// TwinCAT 3 PLC project PLCProgram
// ProgramVersion: 3.1.4026.24
// libraries:
//   FactoryIO_Library, * (Privat)
//   Tc2_ModbusSrv, * (Beckhoff Automation GmbH)
//   Tc2_Standard, * (Beckhoff Automation GmbH)
//   Tc2_System, * (Beckhoff Automation GmbH)
//   Tc2_Utilities, * (Beckhoff Automation GmbH)
// project tree:
//   DUTs/Program/OrderManagement/ OrderData.TcDUT, OrderType.TcDUT
//   DUTs/Program/RFID/ DataPositions.TcDUT
//   DUTs/Program/Warehouse/ StackerCraneStepsLoading.TcDUT, StackerCraneStepsUnloading.TcDUT
//   GVLs/ ConveyorbeltsInfeed.TcGVL, ConveyorbeltsOutfeed.TcGVL, Emitter.TcGVL, GVL.TcGVL, OperatingMode.TcGVL, HMI.TcGVL, OrderManagement.TcGVL, Remover.TcGVL, RFID.TcGVL, Signalmapping.TcGVL, Warehouse.TcGVL
//   / PlcTask.TcTTO
//   POUs/ MAIN.TcPOU, SignalmappingInput.TcPOU, SignalmappingOutput.TcPOU
//   POUs/Programm/AdditionalFunctions/RunControl/ FB_RunControl.TcPOU
//   POUs/Programm/General/ Call_HMI.TcPOU, Call_Operatingmode.TcPOU
//   POUs/Programm/Sections/Infeed/ Call_ConveyorbeltsInfeed.TcPOU, Call_Emitter.TcPOU, Call_RFID.TcPOU
//   POUs/Programm/Sections/Outfeed/ Call_ConveyorbeltsOutfeed.TcPOU, Call_Remover.TcPOU
//   POUs/Programm/Sections/Warehouse/ Call_OrderManagement.TcPOU, Call_Warehouse.TcPOU
// real-time tasks:
//   TASK PlcTask: cycle T#10ms, priority 20, ADS port 350

CONFIGURATION PLCProgram
    RESOURCE PLC ON TwinCAT3
        TASK PlcTask(INTERVAL := T#10ms, PRIORITY := 20);
        PROGRAM MAIN WITH PlcTask : MAIN;
    END_RESOURCE
END_CONFIGURATION

// ---- DUTs/Program/OrderManagement/OrderData.TcDUT
TYPE OrderData :
STRUCT
	JobType	:	OrderType;	//Kind of Order; None, Loading, Unloading
	WarehousePlace	:	WORD;	//Place in the warehouse whre part should be picked or put
	SerialNumberItem	:	WORD;	//Serialnumber of the part
	OrderDone	:	BOOL;	//Current order is finished
	NewOrderSend	:	BOOL;	//Order application has sent new order
	NewOrderReceived	:	BOOL;	//PLC has received new data
END_STRUCT
END_TYPE

// ---- DUTs/Program/OrderManagement/OrderType.TcDUT
{attribute 'qualified_only'}
{attribute 'strict'}
{attribute 'to_string'}
TYPE OrderType :
(
	None := 0,
	Loading,
	Unloading
);
END_TYPE

// ---- DUTs/Program/RFID/DataPositions.TcDUT
TYPE DataPositions :
STRUCT
	FeedInReadingPoint	:	WORD;
	FeedInStackerCrane	:	WORD;
	StackerCraneFork	:	WORD;
END_STRUCT
END_TYPE

// ---- DUTs/Program/Warehouse/StackerCraneStepsLoading.TcDUT
{attribute 'qualified_only'}
{attribute 'strict'}
{attribute 'to_string'}
TYPE StackerCraneStepsLoading :
(
	Waiting := 0,
	DriveToLoadingPosition,
	ForkUnderLoad,
	LiftLoadItem,
	ForkToMiddle,
	DriveToUnloadPrePosition,
	ForkInWarehouse,
	DriveToUnloadPosition
);
END_TYPE

// ---- DUTs/Program/Warehouse/StackerCraneStepsUnloading.TcDUT
{attribute 'qualified_only'}
{attribute 'strict'}
{attribute 'to_string'}
TYPE StackerCraneStepsUnloading :
(
	Waiting := 0,
	DriveToWarehousePlace,
	ForkInWarehouse,
	LiftPart,
	ForkToMiddle,
	DriveToUnloadingPlace,
	ForkToRight,
	LowerPart
);
END_TYPE

// ---- GVLs/ConveyorbeltsInfeed.TcGVL
VAR_GLOBAL
	instConveyorFeedIn	:	FactoryIO.FB_Foerderband;
	instConveyorFeedInStackerCrane	:	FactoryIO.FB_Foerderband;
	conFdIRunControlForwardActiv	:	BOOL;	//Runcontrol forward activ
	conFdIStCRunControlForwardActiv	:	BOOL;	//Runcontrol forward activ
	feConveyorInfeedEnd	:	F_TRIG;	//Falling edge sensor end conveyor infeed
END_VAR

// ---- GVLs/ConveyorbeltsOutfeed.TcGVL
VAR_GLOBAL
	instConveyorFeedOutStackerCrane	:	FactoryIO.FB_Foerderband;
	instConveyorFeedOutTwoMeter	:	FactoryIO.FB_Foerderband;
	instConveyorFeedOutCurve	:	FactoryIO.FB_Foerderband;
	instConveyorFeedOutLong	:	FactoryIO.FB_Foerderband;
	instPartMovingOut	:	FB_RunControl;
END_VAR

// ---- GVLs/Emitter.TcGVL
VAR_GLOBAL
	instEmitterConveyorFeedIn	:	FactoryIO.FB_Emitter;	//Instanz FB_Emitter Zufuehrband Einlauf
	
END_VAR

// ---- GVLs/GVL.TcGVL
{attribute 'qualified_only'}
VAR_GLOBAL
	//Hier die Array-Grenzen anpassen auf die maximale Anzahl an Signalen.
	//Der Name der Liste, darf nicht verändert werden.
	mb_Input_Coils        : ARRAY [0..255] OF BOOL;	//Digital outputs of the PLC
    mb_Output_Coils       : ARRAY [0..255] OF BOOL;	//Digital inputs of the PLC
    mb_Input_Registers    : ARRAY [0..255] OF WORD;	//Analog outputs of the PLC
    mb_Output_Registers   : ARRAY [0..255] OF WORD;	//Analog inputs of the PLC	
END_VAR

// ---- GVLs/OperatingMode.TcGVL
VAR_GLOBAL
	instOperatingmode	:	FactoryIO.FB_OperatingMode;
	currentStateOperatingMode	:	FactoryIO.OperatingMode;
	permissionHardware	:	BOOL := TRUE;
	permissionSafety	:	BOOL := TRUE;
END_VAR

// ---- GVLs/HMI.TcGVL
VAR_GLOBAL
	hmiHeaderInstance	:	FB_HMIHeader;
	hmiHeaderInterface	:	HMIHeader;	
	hmiOperatingmodeInterface	:	HMIInterfaceOperatingMode;
	
	hmiAdsCommunicationInterfaceInstance	:	FB_ADSCommunicationStatus;
	hmiAdsCommunicationInterface	:	ADSCommunicationInterface;
	
	hmiMachineSectionInterface	:	MachineSectionHMIInterface;
	
	hmiEmitterInstances	:	ARRAY[0..0] OF STRING := [
														'FeedIn'
													];
	hmiConveyorInstances	:	ARRAY[0..5] OF STRING := [
															'FeedIn',
															'FeedIn StackerCrane',
															'FeedOut StackerCrane',
															'FeedOut Two meter',
															'FeedOut Curve',
															'FeedOut long'
														 ];
	hmiStackerCraneInstances	:	ARRAY[0..0] OF STRING := [
															'StackerCrane'
														 ];		
	hmiRFIDInstances	:	ARRAY[0..0] OF STRING := [
															'FeedIn StackerCrane'
														 ];
	hmiRemoverInstances	:	ARRAY[0..0] OF STRING := [
														'FeedOut'
													];
END_VAR

// ---- GVLs/OrderManagement.TcGVL
VAR_GLOBAL
	currentOrderData	:	OrderData;
	nextJobReady	:	BOOL;
	reOrderDone	:	R_TRIG;
	reNewOrderSend	:	R_TRIG;
	reShiftSerialNumber	:	R_TRIG;
END_VAR

// ---- GVLs/Remover.TcGVL
VAR_GLOBAL
	ConveyorFeedOutLongRemover	:	BOOL;	//Conveyor feed out long remover
	instRemoverConveyorOutfeedLong	: FactoryIO.FB_Remover;	//Instance of FB_Remover
END_VAR

// ---- GVLs/RFID.TcGVL
VAR_GLOBAL
	instRFIDInfeed	:	FactoryIO.FB_RFID;	//Instance of the RFID-Sensor
	finishedMessageReadSerialNumber	:	BOOL;
	reReadSerialNumber	:	R_TRIG;
	reFinishedMessageReadSerialNumber	:	R_TRIG;
	readData	:	DataPositions;
END_VAR

// ---- GVLs/Signalmapping.TcGVL
VAR_GLOBAL
	BA_Manuel	:	BOOL;	//Operatingmode manual
	BA_Automatik	:	BOOL;	//Operatingmode automatic
	NotAus_Hochregallager	:	BOOL;	//E_Stop
	Start_Automatik_Hochregallager	:	BOOL;	//Automatic Start
	Stop_Automatik_Hochregallager	:	BOOL;	//Automatic Stop
	Grundstellung_Automatik_Hochregallager	:	BOOL;	//Homing
	Reset_Hochregallager	:	BOOL;	//Reset
	Quit_Hochregallager	:	BOOL;	//Quit
	PartPresentConveyorInfeedBegin	:	BOOL;	//Sensor Emitter part present
	PartPresentConveyorInfeedEnd	:	BOOL;	//Sensor conveyor feed in part present
	PartPresentConveyorInfeedStCEnd	:	BOOL;	//Sensor conveyor feed in stacker crane part present
	StackerCraneOneXAxisIsMoving	:	BOOL;	//Stacker crane X axis is moving
	StackerCraneOneZAxisIsMoving	:	BOOL;	//Stacker crane Z axis is moving
	Gabel_InPos_Links	:	BOOL;	//Stacker crane fork in pos left
	Gabel_InPos_Mitte	:	BOOL;	//Stacker crane fork in pos middle
	Gabel_InPos_Rechts	:	BOOL;	//Stacker crane fork in pos right
	SensorConveyorOutfeedStackerCrane	:	BOOL;	//Sensor conveyor feed out stacker crane part present
	SensorConveyorOutfeedEnd	:	BOOL;	//Sensor conveyor feed out part present
	Button_Start_LED	:	BOOL;	//LED start button
	Button_Stop_LED	:	BOOL;	//LED stop button
	Button_Grundstellung_LED	:	BOOL;	//LED homing button
	Button_Reset_LED	:	BOOL;	//LED reset button
	Button_Quit_LED	:	BOOL;	//LED quit button
	EmitterFeedIn	:	BOOL;	//Emitter
	FeedInForward	:	BOOL;	//Conveyor feed in forward
	FeedInStackerCraneForward	:	BOOL;	//Conveyor feed in stacker crane forward
	RFIDFeedInExecuteCommand	:	BOOL;	//RFID feed in stacker crane execute command
	Gabel_zu_Pos_Links	:	BOOL;	//Stacker crane fork left
	Gabel_zu_Pos_Rechts	:	BOOL;	//Stacker crane fork right
	StackerCraneOneLiftFork	:	BOOL;	//Stacker crane lift fork
	ConveyorFeedOutStackerCrane	:	BOOL;	//Conveyor feed out stacker crane forward
	ConveyorFeedOutTwoMeter  	:	BOOL;	//Conveyor feed out forward
	ConveyorCurveFeedOut  	:	BOOL;	//Conveyor curvefeed out forward
	ConveyorFeedOutLong  	:	BOOL;	//Conveyor feed out long forward
	RFIDFeedInReceivedCommandID	:	WORD;	//RFID feed in stacker crane feedback command ID
	RFIDFeedInStatus	:	WORD;	//RFID feed in stacker crane status
	RFIDFeedInReadData	:	WORD;	//RFID feed in stacker crane read data
	RFIDFeedInCommand	:	WORD;	//RFID stacker crane feed in command
	RFIDFeedInMemoryIndex	:	WORD;	//RFID stacker crane feed in memory index
	RFIDFeedInWriteData	:	WORD;	//RFID stacker crane feed in data write
	StackerCraneOneTargetPos  	:	WORD;	//Stacker crane one index position
END_VAR

// ---- GVLs/Warehouse.TcGVL
VAR_GLOBAL
	InUnloading	:	BOOL;
	PartPresent	:	BOOL;
	LoadingSequenceActive	:	BOOL;
	UnloadingSequenceActive	:	BOOL;
	instStackerCrane	:	FB_StackerCrane_Numerical;
	processStepsLoading	: StackerCraneStepsLoading;	
	processStepsUnloading	: StackerCraneStepsUnloading;
	LiftLowerPartLoadingprocess	:	TON;
	LiftLowerPartUnloadingprocess	:	TON;
END_VAR

// ---- POUs/MAIN.TcPOU
PROGRAM MAIN
VAR
	
END_VAR

SignalmappingInput();
Call_Operatingmode();
Call_HMI();
Call_Emitter();
Call_ConveyorbeltsInfeed();
Call_RFID();
Call_OrderManagement();
Call_Warehouse();
Call_ConveyorbeltsOutfeed();
Call_Remover();
SignalmappingOutput();

END_PROGRAM

// ---- POUs/SignalmappingInput.TcPOU
FUNCTION SignalmappingInput

(*=============== Digitale Eingaenge ===============*)
BA_Manuel	:=	GVL.mb_Output_Coils[0];
BA_Automatik	:=	GVL.mb_Output_Coils[1];
NotAus_Hochregallager	:=	GVL.mb_Output_Coils[2];
Start_Automatik_Hochregallager	:=	GVL.mb_Output_Coils[3];
Stop_Automatik_Hochregallager	:=	GVL.mb_Output_Coils[4];
Grundstellung_Automatik_Hochregallager	:=	GVL.mb_Output_Coils[5];
Reset_Hochregallager	:=	GVL.mb_Output_Coils[6];
Quit_Hochregallager	:=	GVL.mb_Output_Coils[7];
PartPresentConveyorInfeedBegin	:=	GVL.mb_Output_Coils[9];
PartPresentConveyorInfeedEnd	:=	GVL.mb_Output_Coils[10];
PartPresentConveyorInfeedStCEnd	:=	GVL.mb_Output_Coils[11];
StackerCraneOneXAxisIsMoving	:=	GVL.mb_Output_Coils[13];
StackerCraneOneZAxisIsMoving	:=	GVL.mb_Output_Coils[14];
Gabel_InPos_Links	:=	GVL.mb_Output_Coils[15];
Gabel_InPos_Rechts	:=	GVL.mb_Output_Coils[16];
Gabel_InPos_Mitte	:=	GVL.mb_Output_Coils[17];
SensorConveyorOutfeedStackerCrane	:=	GVL.mb_Output_Coils[19];
SensorConveyorOutfeedEnd	:=	GVL.mb_Output_Coils[20];

(*=============== Analoge Eingaenge ===============*)
RFIDFeedInReceivedCommandID	:=	GVL.mb_Output_Registers[3];
RFIDFeedInStatus	:=	GVL.mb_Output_Registers[4];
RFIDFeedInReadData	:=	GVL.mb_Output_Registers[5];

END_FUNCTION

// ---- POUs/Programm/General/Call_Operatingmode.TcPOU
FUNCTION Call_Operatingmode

instOperatingmode(PermissionHardware := permissionHardware,
				  PermissionSoftware := permissionSafety,
				  E_Stop := NotAus_Hochregallager,
				  OperatingModeManual:= BA_Manuel, 
				  OperatingModeAutomatic:= BA_Automatik, 
				  HMIInterface := hmiOperatingmodeInterface,
				  LEDStart=> Button_Start_LED, 
				  LEDStop=> Button_Stop_LED, 
				  LEDHome=> Button_Grundstellung_LED, 
				  LEDReset=> Button_Reset_LED, 
				  LEDQuit=> Button_Quit_LED);

instOperatingMode.Start_On(Start_Automatik_Hochregallager);
instOperatingMode.Stop_On(Stop_Automatik_Hochregallager);
instOperatingMode.Homeing_On(Grundstellung_Automatik_Hochregallager);
instOperatingMode.Reset_On(Reset_Hochregallager);
instOperatingMode.Quit_On(Quit_Hochregallager);

currentStateOperatingMode := instOperatingmode.StateOperatingMode;

END_FUNCTION

// ---- POUs/Programm/General/Call_HMI.TcPOU
FUNCTION Call_HMI

hmiHeaderInstance(NameApplication := 'Hochregallager',
				  OperatingModeHMIInterface := hmiOperatingmodeInterface,
				  HeaderHMIInterface := hmiHeaderInterface);
			  
hmiAdsCommunicationInterfaceInstance(Timeout := T#1S,
									 TimeoutHMI := T#500ms,
									 LocalAdsPort := 851,
									 HeartbeatHMI := hmiAdsCommunicationInterface.HeartbeatHMI);
									 

hmiAdsCommunicationInterface.DeviceIpAddress := hmiAdsCommunicationInterfaceInstance.LocalIpAddress;
hmiAdsCommunicationInterface.LocalAMSNetId := hmiAdsCommunicationInterfaceInstance.LocalAMSNetId;
hmiAdsCommunicationInterface.HeartbeatPLC := hmiAdsCommunicationInterfaceInstance.PLCHeartbeatHMICommunication;
hmiAdsCommunicationInterface.RuntimeStatus := hmiAdsCommunicationInterfaceInstance.AdsState;

END_FUNCTION

// ---- POUs/Programm/Sections/Infeed/Call_Emitter.TcPOU
FUNCTION Call_Emitter
VAR_INPUT
END_VAR
VAR
END_VAR

instEmitterConveyorFeedIn(PartPresent:= PartPresentConveyorInfeedBegin, 
					   	  ActorInstanceIndex := 0,
					   	  ActorInstanceName := 'FeedIn',
					   	  HMIInterface := hmiMachineSectionInterface,
					   	  CreatePart=> EmitterFeedIn);
					   
IF NOT PartPresentConveyorInfeedBegin AND 
	currentStateOperatingMode.AutomaticStart.IsActive
THEN
	instEmitterConveyorFeedIn.Create();
END_IF

END_FUNCTION

// ---- POUs/Programm/Sections/Infeed/Call_ConveyorbeltsInfeed.TcPOU
FUNCTION Call_ConveyorbeltsInfeed

(*================ FeedIn ================*)
instConveyorFeedIn(
	SensorInfeed:= PartPresentConveyorInfeedBegin, 
	SensorOutfeed:= PartPresentConveyorInfeedEnd, 
	MaximumTimeRuncontrol:= T#30S, 
	ActorInstanceIndex := 0,
	ActorInstanceName := 'FeedIn',
	HMIInterface := hmiMachineSectionInterface,
	MotorForward=> FeedInForward, 
	RuncontrolForwardActive=> conFdIRunControlForwardActiv, 
	OperatingMode:= instOperatingMode.StateOperatingMode);
	
instConveyorFeedIn.MotorForward_On((PartPresentConveyorInfeedBegin OR conFdIRunControlForwardActiv OR
									(PartPresentConveyorInfeedEnd AND finishedMessageReadSerialNumber)) 
											AND NOT PartPresentConveyorInfeedStCEnd AND Gabel_InPos_Mitte);
instConveyorFeedIn.Motor_Off(PartPresentConveyorInfeedEnd AND NOT finishedMessageReadSerialNumber);

(*================ FeedIn Stacker Crane ================*)
instConveyorFeedInStackerCrane(
	SensorInfeed:= PartPresentConveyorInfeedEnd, 
	SensorOutfeed:= PartPresentConveyorInfeedStCEnd, 
	MaximumTimeRuncontrol:= T#30S,  
	ActorInstanceIndex := 1,
	ActorInstanceName := 'FeedIn Stacker Crane',
	HMIInterface := hmiMachineSectionInterface,
	MotorForward=> FeedInStackerCraneForward, 
	RuncontrolForwardActive=> conFdIStCRunControlForwardActiv, 
	OperatingMode:= instOperatingMode.StateOperatingMode);
	
instConveyorFeedInStackerCrane.MotorForward_On(PartPresentConveyorInfeedEnd AND NOT PartPresentConveyorInfeedStCEnd
									AND Gabel_InPos_Mitte AND finishedMessageReadSerialNumber);
instConveyorFeedInStackerCrane.Motor_Off(PartPresentConveyorInfeedStCEnd);

(*================ Data shifting ================*)
feConveyorInfeedEnd(CLK := PartPresentConveyorInfeedEnd);
IF feConveyorInfeedEnd.Q THEN
	readData.FeedInStackerCrane := readData.FeedInReadingPoint;
	//readData.FeedInReadingPoint := 0;
END_IF

END_FUNCTION

// ---- POUs/Programm/Sections/Infeed/Call_RFID.TcPOU
FUNCTION Call_RFID

instRFIDInfeed(PermissionHardware := permissionHardware,
		   	   QuitError := instOperatingMode.StateOperatingMode.Quit.IsActive,
		   	   Reset := instOperatingMode.StateOperatingMode.Reset.IsActive,
		   	   SensorPartDetected := PartPresentConveyorInfeedEnd,
		   	   CommandID := RFIDFeedInReceivedCommandID,
		   	   ReadData := RFIDFeedInReadData,
		   	   Status := RFIDFeedInStatus,
		   	   ActorInstanceIndex := 0,
		   	   ActorInstanceName := 'FeedIn StackerCrane',
		   	   HMIInterface := HMI.hmiMachineSectionInterface,
		   	   FMReadingSerialNumber => finishedMessageReadSerialNumber,
		   	   ExecuteCommand => RFIDFeedInExecuteCommand,
		   	   Command => RFIDFeedInCommand,
		   	   WriteData => RFIDFeedInWriteData,
		   	   MemoryIndex => RFIDFeedInMemoryIndex);

reReadSerialNumber(CLK := PartPresentConveyorInfeedEnd AND NOT finishedMessageReadSerialNumber);			   
reFinishedMessageReadSerialNumber(CLK := finishedMessageReadSerialNumber);
instRFIDInfeed.ReadSerialNumber(reReadSerialNumber.Q);

IF reFinishedMessageReadSerialNumber.Q THEN
	readData.FeedInReadingPoint := RFIDFeedInReadData;
END_IF

END_FUNCTION

// ---- POUs/Programm/Sections/Warehouse/Call_OrderManagement.TcPOU
FUNCTION Call_OrderManagement

reNewOrderSend(CLK := currentOrderData.NewOrderSend);

IF reNewOrderSend.Q THEN
	currentOrderData.NewOrderReceived := TRUE;
END_IF

reOrderDone(CLK := currentOrderData.OrderDone);

IF reOrderDone.Q THEN
	currentOrderData.JobType := OrderType.None;
	currentOrderData.SerialNumberItem := 0;
	currentOrderData.WarehousePlace := 0;
	currentOrderData.OrderDone := FALSE;
END_IF

nextJobReady := currentOrderData.JobType <> OrderType.None AND
				currentOrderData.WarehousePlace <> 0 AND NOT
				currentOrderData.OrderDone;

END_FUNCTION

// ---- POUs/Programm/Sections/Warehouse/Call_Warehouse.TcPOU
FUNCTION Call_Warehouse

instStackerCrane(XAxisMoving := StackerCraneOneXAxisIsMoving,
				 ZAxisMoving := StackerCraneOneZAxisIsMoving,
				 ActorInstanceIndex := 0,
				 ActorInstanceName := 'Zufuehrung',
				 ForkInPosLeft := Gabel_InPos_Links,
				 ForkInPosMiddle := Gabel_InPos_Mitte,
				 ForkInPosRight := Gabel_InPos_Rechts,
				 OperatingMode := instOperatingMode.StateOperatingMode,
				 HMIInterface := HMI.hmiMachineSectionInterface,
				 LiftFork => StackerCraneOneLiftFork,
				 MoveForkLeft => Gabel_zu_Pos_Links,
				 MoveForkRight => Gabel_zu_Pos_Rechts,
				 TargetPos => StackerCraneOneTargetPos);
				 
(*================ Steps ================*)
IF instOperatingMode.StateOperatingMode.Reset.IsActive THEN
	processStepsLoading := StackerCraneStepsLoading.Waiting;
END_IF

CASE processStepsLoading OF
	StackerCraneStepsLoading.Waiting:
		instStackerCrane.MoveForkToMiddle_ON(TRUE);
		IF instOperatingMode.StateOperatingMode.AutomaticStart.IsActive AND nextJobReady
			AND currentOrderData.JobType = OrderType.Loading
		THEN
			processStepsLoading := StackerCraneStepsLoading.DriveToLoadingPosition;
		END_IF
StackerCraneStepsLoading.DriveToLoadingPosition:
		instStackerCrane.MoveAxesStackerCrane_ON(TRUE, 55);	
		IF instStackerCrane.InPositionXAxis AND instStackerCrane.InPositionZAxis
		AND NOT instStackerCrane.NewOrderActive AND PartPresentConveyorInfeedStCEnd
		THEN
			InUnloading	:= FALSE;
			processStepsLoading := StackerCraneStepsLoading.ForkUnderLoad;
		END_IF
StackerCraneStepsLoading.ForkUnderLoad:
		InUnloading	:= FALSE;
		instStackerCrane.MoveForkToLeft_ON(TRUE);
		IF Gabel_InPos_Links THEN
			processStepsLoading := StackerCraneStepsLoading.LiftLoadItem;
		END_IF
StackerCraneStepsLoading.LiftLoadItem:
		instStackerCrane.MoveForkToLeft_ON(TRUE);
		instStackerCrane.LiftForkUp(TRUE);
		IF instStackerCrane.InPositionXAxis AND instStackerCrane.InPositionZAxis
		THEN
			processStepsLoading := StackerCraneStepsLoading.ForkToMiddle;
		END_IF
StackerCraneStepsLoading.ForkToMiddle:
		instStackerCrane.MoveForkToMiddle_ON(TRUE);
		IF Gabel_InPos_Mitte AND NOT InUnloading THEN
			processStepsLoading := StackerCraneStepsLoading.DriveToUnloadPrePosition;
		ELSIF Gabel_InPos_Mitte AND InUnloading THEN
			currentOrderData.OrderDone := TRUE;
			processStepsLoading := StackerCraneStepsLoading.Waiting;
		END_IF
StackerCraneStepsLoading.DriveToUnloadPrePosition:
		instStackerCrane.MoveAxesStackerCrane_ON(TRUE, currentOrderData.WarehousePlace);
		IF instStackerCrane.InPositionXAxis AND instStackerCrane.InPositionZAxis
		AND NOT instStackerCrane.NewOrderActive
		THEN
			processStepsLoading := StackerCraneStepsLoading.ForkInWarehouse;
		END_IF
StackerCraneStepsLoading.ForkInWarehouse:
		instStackerCrane.MoveForkToRight_ON(TRUE);
		IF Gabel_InPos_Rechts THEN
			processStepsLoading := StackerCraneStepsLoading.DriveToUnloadPosition;
		END_IF
StackerCraneStepsLoading.DriveToUnloadPosition:
		instStackerCrane.MoveForkToRight_ON(TRUE);
		instStackerCrane.LowerForkUp(TRUE);
		IF instStackerCrane.InPositionXAxis AND instStackerCrane.InPositionZAxis
		THEN
			InUnloading	:= TRUE;
			processStepsLoading := StackerCraneStepsLoading.ForkToMiddle;
		END_IF
END_CASE

(*================ Data shifting ================*)
reShiftSerialNumber(CLK := processStepsLoading = StackerCraneStepsLoading.LiftLoadItem);
IF reShiftSerialNumber.Q THEN
	readData.StackerCraneFork := readData.FeedInStackerCrane;
	currentOrderData.SerialNumberItem := readData.StackerCraneFork;
END_IF

END_FUNCTION

// ---- POUs/Programm/Sections/Outfeed/Call_ConveyorbeltsOutfeed.TcPOU
FUNCTION Call_ConveyorbeltsOutfeed

(*================ Runcontrol ================*)
instPartMovingOut.ActivateRunControl(SensorConveyorOutfeedStackerCrane AND Gabel_InPos_Mitte);
instPartMovingOut.DeactivateRunControl(SensorConveyorOutfeedEnd);

(*================ FeedOut Stacker Crane ================*)
instConveyorFeedOutStackerCrane(  
	SensorOutfeed:= TRUE,
	MaximumTimeRuncontrol:= T#30S, 
	ActorInstanceIndex := 2,
	ActorInstanceName := 'FeedOut StackerCrane',
	HMIInterface := hmiMachineSectionInterface,
	OperatingMode:= instOperatingMode.StateOperatingMode,
	MotorForward=> ConveyorFeedOutStackerCrane);
	
instConveyorFeedOutStackerCrane.MotorForward_On(instPartMovingOut.IsActive);
instConveyorFeedOutStackerCrane.Motor_Off(NOT instPartMovingOut.IsActive AND NOT instOperatingmode.StateOperatingMode.ManuelIsActive);

(*================ FeedOut Two Meter ================*)
instConveyorFeedOutTwoMeter(  
	SensorOutfeed:= TRUE,
	MaximumTimeRuncontrol:= T#30S,  
	ActorInstanceIndex := 3,
	ActorInstanceName := 'FeedOut Two meter',
	HMIInterface := hmiMachineSectionInterface, 
	OperatingMode:= instOperatingMode.StateOperatingMode,
	MotorForward=> ConveyorFeedOutTwoMeter);
	
instConveyorFeedOutTwoMeter.MotorForward_On(instPartMovingOut.IsActive);
instConveyorFeedOutTwoMeter.Motor_Off(NOT instPartMovingOut.IsActive AND NOT instOperatingmode.StateOperatingMode.ManuelIsActive);

(*================ FeedOut Curve ================*)
instConveyorFeedOutCurve(  
	SensorOutfeed:= TRUE,
	MaximumTimeRuncontrol:= T#30S,  
	ActorInstanceIndex := 4,
	ActorInstanceName := 'FeedOut Curve',
	HMIInterface := hmiMachineSectionInterface, 
	OperatingMode:= instOperatingMode.StateOperatingMode,
	MotorForward=> ConveyorCurveFeedOut);
	
instConveyorFeedOutCurve.MotorForward_On(instPartMovingOut.IsActive);
instConveyorFeedOutCurve.Motor_Off(NOT instPartMovingOut.IsActive AND NOT instOperatingmode.StateOperatingMode.ManuelIsActive);

(*================ FeedOut Long ================*)
instConveyorFeedOutLong(  
	SensorOutfeed:= TRUE,
	MaximumTimeRuncontrol:= T#30S,  
	ActorInstanceIndex := 5,
	ActorInstanceName := 'FeedOut Long',
	HMIInterface := hmiMachineSectionInterface, 
	OperatingMode:= instOperatingMode.StateOperatingMode,
	MotorForward=> ConveyorFeedOutLong);
	
instConveyorFeedOutLong.MotorForward_On(instPartMovingOut.IsActive);
instConveyorFeedOutLong.Motor_Off(NOT instPartMovingOut.IsActive AND NOT instOperatingmode.StateOperatingMode.ManuelIsActive);

END_FUNCTION

// ---- POUs/Programm/Sections/Outfeed/Call_Remover.TcPOU
FUNCTION Call_Remover

instRemoverConveyorOutfeedLong(PartPresent:= SensorConveyorOutfeedEnd, 
					   	  	   ActorInstanceIndex := 0,
					   	  	   ActorInstanceName := 'FeedOut',
					   	  	   HMIInterface := hmiMachineSectionInterface,
						  	   OperatingModeSection := instOperatingMode.StateOperatingMode,
					   	  	   RemovePart=> ConveyorFeedOutLongRemover);

instRemoverConveyorOutfeedLong.Remove();

END_FUNCTION

// ---- POUs/SignalmappingOutput.TcPOU
FUNCTION SignalmappingOutput

(*=============== Digitale Ausgaenge ===============*)
GVL.mb_Input_Coils[3]	:=	Button_Start_LED;
GVL.mb_Input_Coils[4]	:=	Button_Stop_LED;
GVL.mb_Input_Coils[5]	:=	Button_Grundstellung_LED;
GVL.mb_Input_Coils[6]	:=	Button_Reset_LED;
GVL.mb_Input_Coils[7]	:=	Button_Quit_LED;
GVL.mb_Input_Coils[9]	:=	EmitterFeedIn;
GVL.mb_Input_Coils[10]	:=	FeedInForward;
GVL.mb_Input_Coils[11]	:=	FeedInStackerCraneForward;
GVL.mb_Input_Coils[12]	:=	RFIDFeedInExecuteCommand;
GVL.mb_Input_Coils[15]	:=	Gabel_zu_Pos_Links;
GVL.mb_Input_Coils[16]	:=	Gabel_zu_Pos_Rechts;
GVL.mb_Input_Coils[17]	:=	StackerCraneOneLiftFork;
GVL.mb_Input_Coils[19]	:=	ConveyorFeedOutStackerCrane;
GVL.mb_Input_Coils[20]	:=	ConveyorFeedOutTwoMeter;
GVL.mb_Input_Coils[21]	:=	ConveyorCurveFeedOut;
GVL.mb_Input_Coils[22]	:=	ConveyorFeedOutLong;
GVL.mb_Input_Coils[23]	:=	ConveyorFeedOutLongRemover;

(*=============== Analoge Ausgaenge ===============*)
GVL.mb_Input_Registers[3]	:=	RFIDFeedInCommand;
GVL.mb_Input_Registers[4]	:=	RFIDFeedInMemoryIndex;
GVL.mb_Input_Registers[5]	:=	RFIDFeedInWriteData;
GVL.mb_Input_Registers[7]	:=	StackerCraneOneTargetPos;

END_FUNCTION

// ---- POUs/Programm/AdditionalFunctions/RunControl/FB_RunControl.TcPOU
FUNCTION_BLOCK PUBLIC FB_RunControl
VAR
	statRuncontrolActive	:	BOOL;
END_VAR

METHOD PUBLIC ActivateRunControl
VAR_INPUT
	Activate	:	BOOL;
END_VAR
IF Activate	THEN
	statRuncontrolActive := TRUE;
END_IF
END_METHOD

METHOD PUBLIC DeactivateRunControl
VAR_INPUT
	Deactivate	:	BOOL;
END_VAR
IF Deactivate THEN
	statRuncontrolActive := FALSE;
END_IF
END_METHOD

PROPERTY PUBLIC IsActive : BOOL
GET
IsActive := statRuncontrolActive;
END_GET
END_PROPERTY

END_FUNCTION_BLOCK
